SYSTEM nameless
  (* Version 1.0 *)
  APPLICATION namelessApp
    FBS
      E_PERMIT_2 : E_PERMIT(PERMIT := None);
      E_PERMIT_3 : E_PERMIT(PERMIT := None);
      E_PERMIT_1 : E_PERMIT(PERMIT := None);
      E_PERMIT : E_PERMIT(PERMIT := None);
      E_SPLIT : E_SPLIT;
      E_CTU : E_CTU(PV := None, Q := None, CV := None);
      E_RESTART : E_RESTART;
    END_FBS
    EVENT_CONNECTIONS
      E_PERMIT_2.EO TO E_CTU.R;
      E_PERMIT.EO TO E_SPLIT.EI;
      E_SPLIT.EO1 TO E_CTU.CU;
      E_SPLIT.EO2 TO E_PERMIT_1.EI;
      E_CTU.CUO TO E_PERMIT_2.EI;
      E_CTU.RO TO E_PERMIT_3.EI;
      E_RESTART.WARM TO E_PERMIT.EI;
    END_CONNECTIONS
    DATA_CONNECTIONS
      E_CTU.Q TO E_PERMIT_2.PERMIT;
    END_CONNECTIONS
  END_APPLICATION
END_SYSTEM
